(* PLC project benzene-distillation, Generated TextualNotationConverter 1.0 *)
(* stored: creationDateTime 2025-07-30T12:00:00, modificationDateTime 2025-01-30T12:00:00 *)

FUNCTION_BLOCK ANALOG_IN
  VAR_INPUT
    Name : STRING;
    Description : STRING;
    Raw_Signal : REAL;
    PV_High : REAL;
    PV_Low : REAL;
    Scaling_Slope : REAL;
    Scaling_Offset : REAL;
    Alarm_Enable : BOOL;
  END_VAR
  VAR_OUTPUT
    PV : REAL;
    High_Alarm : BOOL;
    Low_Alarm : BOOL;
    General_Fault : BOOL;
  END_VAR

            
          
END_FUNCTION_BLOCK

FUNCTION_BLOCK DIGITAL_IN
  VAR_INPUT
    Name : STRING;
    Description : STRING;
    DI_Raw : BOOL;
    DebounceTime : STRING;
    EnableAlarm : BOOL;
  END_VAR
  VAR_OUTPUT
    DI_Out : BOOL;
    Fault_State : BOOL;
  END_VAR

            
          
END_FUNCTION_BLOCK

FUNCTION_BLOCK PID_BASIC
  VAR_INPUT
    Name : STRING;
    Description : STRING;
    AUTO : BOOL;
    PV : REAL;
    SP : REAL;
    MV_MIN : REAL;
    MV_MAX : REAL;
    X0 : REAL;
    KP : REAL;
    TR : REAL;
    TD : REAL;
    PV_High : REAL;
    PV_Low : REAL;
    Deviation_Limit : REAL;
    Inhibit : BOOL;
  END_VAR
  VAR_OUTPUT
    PV_High_Alarm : BOOL;
    PV_Low_Alarm : BOOL;
    Deviation_Alarm : BOOL;
    XOUT : REAL;
  END_VAR

            
          
END_FUNCTION_BLOCK

FUNCTION_BLOCK VALVE_ELECTRIC
  VAR_INPUT
    Name : STRING;
    Description : STRING;
    Control_Signal : REAL;
    Manual_Mode : BOOL;
    Manual_Position : REAL;
    Open_Limit : REAL;
    Close_Limit : REAL;
    Timeout : STRING;
    Inhibit : BOOL;
  END_VAR
  VAR_OUTPUT
    Valve_Position : REAL;
    Feedback_Pos : REAL;
    Valve_Moving : BOOL;
    Position_Error : BOOL;
    Alarm : BOOL;
  END_VAR

            
          
END_FUNCTION_BLOCK

FUNCTION_BLOCK VALVE_ON_OFF
  VAR_INPUT
    Name : STRING;
    Description : STRING;
    Open_Cmd : BOOL;
    Close_Cmd : BOOL;
    Timeout : STRING;
    Inhibit : BOOL;
  END_VAR
  VAR_OUTPUT
    FB_Opened : BOOL;
    FB_Closed : BOOL;
    Valve_Open_Out : BOOL;
    Valve_Close_Out : BOOL;
    Alarm_Position_Error : BOOL;
    Alarm_General : BOOL;
  END_VAR

            
          
END_FUNCTION_BLOCK

PROGRAM Section2
  VAR
    TE101_Temperature_PV : REAL;
    LIT101_Level_PV : REAL;
    PIT102_Pressure_PV : REAL;
    TIC104_MV_Percent : REAL;
    PV103_Position_FB : REAL;
  END_VAR
  VAR
    TE-101 : ANALOG_IN;
    LIT-101 : ANALOG_IN;
    PIT-102 : ANALOG_IN;
    TIC-104 : PID_BASIC;
    PV-103 : VALVE_ELECTRIC;
    XV-105 : VALVE_ON_OFF;
    LAH-101 : DIGITAL_IN;
    LAL-101 : DIGITAL_IN;
  END_VAR

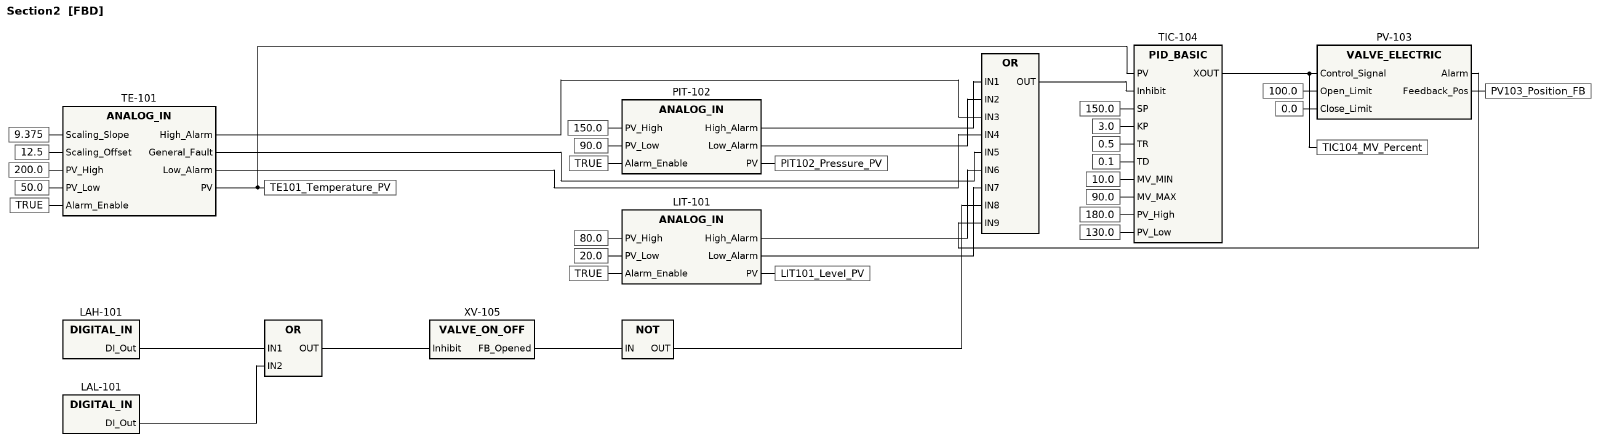
(* FBD diagram, written out as Structured Text *)
LIT-101(PV_High := 80.0, PV_Low := 20.0, Alarm_Enable := TRUE);
LIT101_Level_PV := LIT-101.PV;
PIT-102(PV_High := 150.0, PV_Low := 90.0, Alarm_Enable := TRUE);
PIT102_Pressure_PV := PIT-102.PV;
TE-101(Scaling_Slope := 9.375, Scaling_Offset := 12.5, PV_High := 200.0, PV_Low := 50.0, Alarm_Enable := TRUE);
LAH-101();
LAL-101();
XV-105(Inhibit := LAH-101.DI_Out OR LAL-101.DI_Out);
TIC-104(PV := TE-101.PV, Inhibit := PIT-102.High_Alarm OR PIT-102.Low_Alarm OR TE-101.High_Alarm OR TE-101.Low_Alarm OR TE-101.General_Fault OR LIT-101.High_Alarm OR LIT-101.Low_Alarm OR NOT XV-105.FB_Opened OR PV-103.Alarm, SP := 150.0, KP := 3.0, TR := 0.5, TD := 0.1, MV_MIN := 10.0, MV_MAX := 90.0, PV_High := 180.0, PV_Low := 130.0);
PV-103(Control_Signal := TIC-104.XOUT, Open_Limit := 100.0, Close_Limit := 0.0);
PV103_Position_FB := PV-103.Feedback_Pos;
TE101_Temperature_PV := TE-101.PV;
TIC104_MV_Percent := TIC-104.XOUT;
END_PROGRAM

FUNCTION_BLOCK BOOL_IN
  VAR_INPUT
    Name : STRING;
    Description : STRING;
    Bool_In : BOOL;
    Alarm_OnTrue : BOOL;
    Alarm_OnFalse : BOOL;
    Latch_Enable : BOOL;
    Reset_Latch : BOOL;
  END_VAR
  VAR_OUTPUT
    Bool_Out : BOOL;
    Alarm_Active : BOOL;
    Latched_Status : BOOL;
  END_VAR

            
          
END_FUNCTION_BLOCK

FUNCTION_BLOCK DUTY_STANDBY
  VAR_INPUT
    Name : STRING;
    Description : STRING;
    Enable : BOOL;
    StartRequest : BOOL;
    AlternateEnable : BOOL;
    ForcePumpA : BOOL;
    ForcePumpB : BOOL;
    DutyElapsed : BOOL;
    MinRunElapsed : BOOL;
    SwitchoverDelayElapsed : BOOL;
    StartTimeoutElapsed : BOOL;
    PumpA_RunFB : BOOL;
    PumpB_RunFB : BOOL;
    PumpA_Fault : BOOL;
    PumpB_Fault : BOOL;
    Reset : BOOL;
    Inhibit : BOOL;
  END_VAR
  VAR_OUTPUT
    CmdPumpA : BOOL;
    CmdPumpB : BOOL;
    ActiveIsA : BOOL;
    SwitchedDueToDuty : BOOL;
    SwitchedDueToFailure : BOOL;
    Alarm_FailedStart_A : BOOL;
    Alarm_FailedStart_B : BOOL;
    Alarm_NoAvailablePump : BOOL;
  END_VAR

            
          
END_FUNCTION_BLOCK

FUNCTION_BLOCK MOTOR_2SPD
  VAR_INPUT
    Name : STRING;
    Description : STRING;
    Start_Cmd : BOOL;
    Stop_Cmd : BOOL;
    Speed_High_Cmd : BOOL;
    Speed_Low_Cmd : BOOL;
    Inhibit : BOOL;
  END_VAR
  VAR_OUTPUT
    Motor_Start_Out : BOOL;
    FB_Running : BOOL;
    FB_Trip : BOOL;
    FB_HighSpeed : BOOL;
    FB_LowSpeed : BOOL;
    Alarm_Speed_Error : BOOL;
  END_VAR

            
          
END_FUNCTION_BLOCK

FUNCTION_BLOCK MOTOR_ON_OFF
  VAR_INPUT
    Name : STRING;
    Description : STRING;
    Start_Cmd : BOOL;
    Stop_Cmd : BOOL;
    Start_Delay : STRING;
    MinRunTime : STRING;
    Inhibit : BOOL;
  END_VAR
  VAR_OUTPUT
    Motor_Start_Out : BOOL;
    FB_Running : BOOL;
    FB_Trip : BOOL;
    Alarm_Start_Fail : BOOL;
    Alarm_Stop_Fail : BOOL;
  END_VAR

            
          
END_FUNCTION_BLOCK

FUNCTION_BLOCK MOTOR_VSD
  VAR_INPUT
    Name : STRING;
    Description : STRING;
    Start_Cmd : BOOL;
    Stop_Cmd : BOOL;
    Speed_SP : REAL;
    Accel_Ramp : STRING;
    Decel_Ramp : STRING;
    Inhibit : BOOL;
  END_VAR
  VAR_OUTPUT
    Speed_Out : REAL;
    FB_Running : BOOL;
    FB_Fault : BOOL;
    FB_Ready : BOOL;
    FB_ActualSpeed : REAL;
    Alarm_Speed_Deviation : BOOL;
    Alarm_Comm_Fail : BOOL;
  END_VAR

            
          
END_FUNCTION_BLOCK

FUNCTION_BLOCK RATIO_CONTROL
  VAR_INPUT
    Name : STRING;
    Description : STRING;
    Auto : BOOL;
    PrimaryPV : REAL;
    SecondaryPV : REAL;
    RatioSP : REAL;
    Bias : REAL;
    TrimKp : REAL;
    TrimTi : STRING;
    MV_MIN : REAL;
    MV_MAX : REAL;
    ManOut : REAL;
    Inhibit : BOOL;
  END_VAR
  VAR_OUTPUT
    SlaveSP : REAL;
    ActiveRatio : REAL;
    RatioErr : REAL;
  END_VAR

            
          
END_FUNCTION_BLOCK

FUNCTION_BLOCK SPLIT_RANGE
  VAR_INPUT
    Name : STRING;
    Description : STRING;
    IN : REAL;
    Split_Point : REAL;
    Output1_Start : REAL;
    Output1_End : REAL;
    Output2_Start : REAL;
    Output2_End : REAL;
  END_VAR
  VAR_OUTPUT
    OUT1 : REAL;
    OUT2 : REAL;
  END_VAR

            
          
END_FUNCTION_BLOCK

FUNCTION_BLOCK VOTING_ANALOG
  VAR_INPUT
    Name : STRING;
    Description : STRING;
    Input1 : REAL;
    Input2 : REAL;
    Input3 : REAL;
    Deviation_Limit : REAL;
    Voting_Scheme : STRING;
    EnableAlarm : BOOL;
    Inhibit : BOOL;
  END_VAR
  VAR_OUTPUT
    Voted_Output : REAL;
    Sensor1_Fault : BOOL;
    Sensor2_Fault : BOOL;
    Sensor3_Fault : BOOL;
    Alarm_Voting_Error : BOOL;
    Healthy_Sensors_Count : INT;
  END_VAR

            
          
END_FUNCTION_BLOCK

PROGRAM Section3
  VAR
    Reboiler_Temperature_PV_TI106 : REAL;
    Steam_Flow_PV_FIT101 : REAL;
    Column_Pressure_PV_PT101 : REAL;
    FIC104_MV_SteamValveCmd : REAL;
    LIC002_LowLevel_Trip : BOOL;
  END_VAR
  VAR
    TI-106 : ANALOG_IN;
    FIT-101 : ANALOG_IN;
    PT-101 : ANALOG_IN;
    FIC-104 : PID_BASIC;
    TCV-106 : VALVE_ELECTRIC;
    LIC-002 : BOOL_IN;
    TAH-106 : BOOL_IN;
    TAL-106 : BOOL_IN;
    FAH-104 : BOOL_IN;
  END_VAR
  VAR  (* added by the conversion: wires and edge detectors of the diagram *)
    _OR38_OUT : BOOL;
  END_VAR

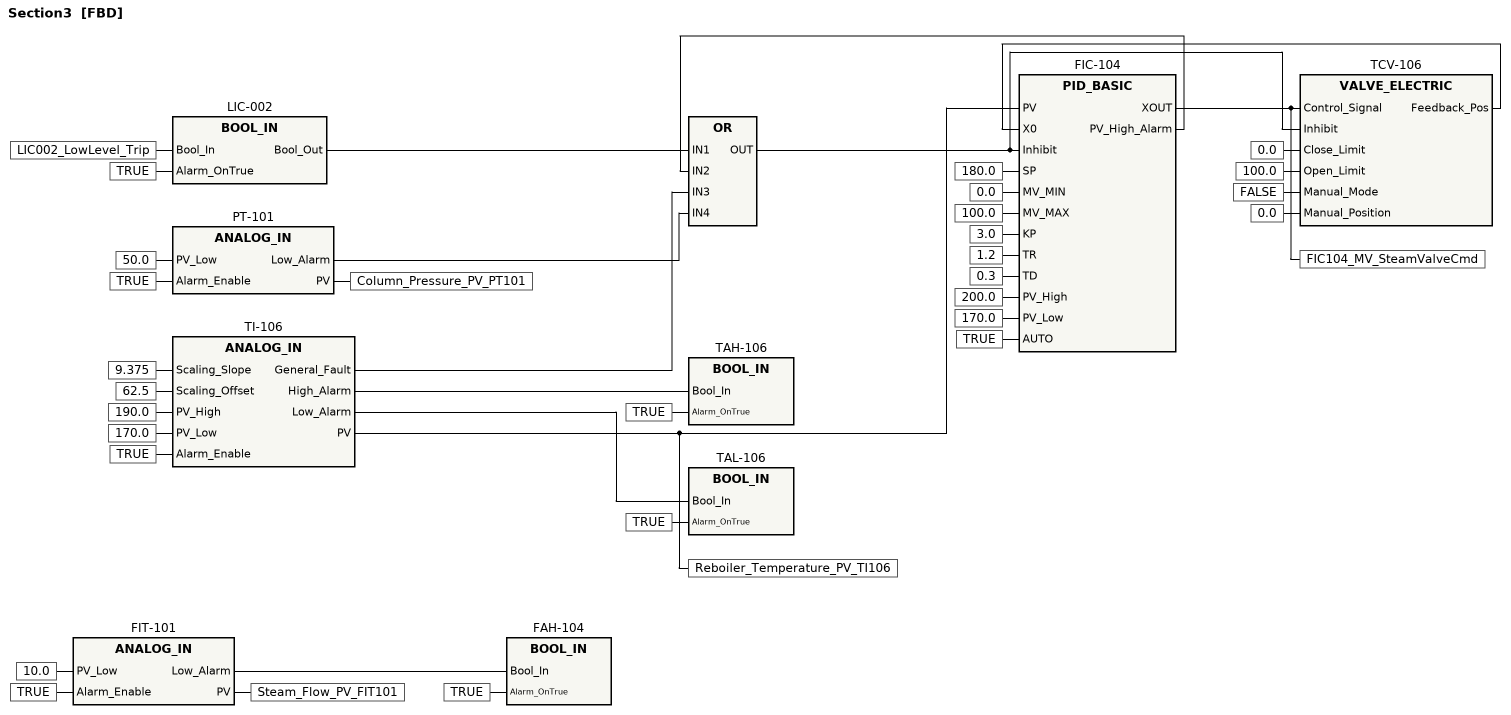
(* FBD diagram, written out as Structured Text *)
PT-101(PV_Low := 50.0, Alarm_Enable := TRUE);
Column_Pressure_PV_PT101 := PT-101.PV;
TI-106(Scaling_Slope := 9.375, Scaling_Offset := 62.5, PV_High := 190.0, PV_Low := 170.0, Alarm_Enable := TRUE);
LIC-002(Bool_In := LIC002_LowLevel_Trip, Alarm_OnTrue := TRUE);
_OR38_OUT := LIC-002.Bool_Out OR FIC-104.PV_High_Alarm OR TI-106.General_Fault OR PT-101.Low_Alarm;
TCV-106(Control_Signal := FIC-104.XOUT, Inhibit := _OR38_OUT, Close_Limit := 0.0, Open_Limit := 100.0, Manual_Mode := FALSE, Manual_Position := 0.0);
FIC-104(PV := TI-106.PV, X0 := TCV-106.Feedback_Pos, Inhibit := _OR38_OUT, SP := 180.0, MV_MIN := 0.0, MV_MAX := 100.0, KP := 3.0, TR := 1.2, TD := 0.3, PV_High := 200.0, PV_Low := 170.0, AUTO := TRUE);
FIC104_MV_SteamValveCmd := FIC-104.XOUT;
Reboiler_Temperature_PV_TI106 := TI-106.PV;
FIT-101(PV_Low := 10.0, Alarm_Enable := TRUE);
Steam_Flow_PV_FIT101 := FIT-101.PV;
TAH-106(Bool_In := TI-106.High_Alarm, Alarm_OnTrue := TRUE);
TAL-106(Bool_In := TI-106.Low_Alarm, Alarm_OnTrue := TRUE);
FAH-104(Bool_In := FIT-101.Low_Alarm, Alarm_OnTrue := TRUE);
END_PROGRAM

PROGRAM Section4
  VAR
    LT_105_Level_PV : REAL;
    FT_107_Flow_PV : REAL;
    PT_104_Pressure_PV : REAL;
    LIC_104_RSP_to_FIC_107_GPM : REAL;
    FIC_107_Control_Signal_to_LV_107 : REAL;
    XV103_NotOpen : BOOL;
    Cascade_Inhibit : BOOL;
    Permissive_OK : BOOL;
  END_VAR
  VAR
    LT-105 : ANALOG_IN;
    FT-107 : ANALOG_IN;
    PT-104 : ANALOG_IN;
    LIC-104 : PID_BASIC;
    FIC-107 : PID_BASIC;
    PIC-104 : PID_BASIC;
    LV-107 : VALVE_ELECTRIC;
    XV-103 : VALVE_ON_OFF;
  END_VAR
  VAR  (* added by the conversion: wires and edge detectors of the diagram *)
    _NOT80_OUT : BOOL;
    _OR79_OUT : BOOL;
    _MULT83_OUT : REAL;
  END_VAR

(* FBD diagram, written out as Structured Text *)
XV-103();
_NOT80_OUT := NOT XV-103.FB_Opened;
LT-105(PV_High := 90.0, PV_Low := 10.0, Alarm_Enable := TRUE);
PT-104(PV_High := 30.0, PV_Low := 15.0, Alarm_Enable := TRUE);
FT-107(PV_High := 50.0, PV_Low := 0.0, Alarm_Enable := TRUE);
LIC-104(PV := LT-105.PV, Inhibit := _OR79_OUT, AUTO := TON(NOT _OR79_OUT, T#30s), SP := 65.0, KP := 1.5, TR := 2.5, TD := 0.0, MV_MIN := 0.0, MV_MAX := 100.0, X0 := 40.0, PV_High := 90.0, PV_Low := 10.0);
_MULT83_OUT := MULT(LIC-104.XOUT, 0.5);
FIC-107(SP := _MULT83_OUT, PV := FT-107.PV, Inhibit := _OR79_OUT, AUTO := NOT _OR79_OUT, KP := 4.0, TR := 0.5, TD := 0.0, MV_MIN := 0.0, MV_MAX := 100.0, PV_High := 50.0, PV_Low := 0.0);
LV-107(Control_Signal := FIC-107.XOUT, Inhibit := PT-104.High_Alarm, Manual_Mode := PT-104.High_Alarm, Open_Limit := 100.0, Close_Limit := 0.0, Manual_Position := 0.0);
_OR79_OUT := _NOT80_OUT OR LT-105.Low_Alarm OR PT-104.Low_Alarm OR PT-104.High_Alarm OR FT-107.General_Fault OR LV-107.Alarm;
Cascade_Inhibit := _OR79_OUT;
FIC_107_Control_Signal_to_LV_107 := FIC-107.XOUT;
FT_107_Flow_PV := FT-107.PV;
LIC_104_RSP_to_FIC_107_GPM := _MULT83_OUT;
LT_105_Level_PV := LT-105.PV;
PT_104_Pressure_PV := PT-104.PV;
Permissive_OK := NOT _OR79_OUT;
XV103_NotOpen := _NOT80_OUT;
PIC-104(PV := PT-104.PV);
END_PROGRAM

PROGRAM Section5
  VAR
    FI102_FlowRate : REAL;
    PI102_Pressure : REAL;
    LCV102_PositionCmd : REAL;
    XV102A_OpenCmd : BOOL;
    XV102A_CloseCmd : BOOL;
    XV102B_OpenCmd : BOOL;
    XV102B_CloseCmd : BOOL;
    XV102A_OpenFB : BOOL;
    XV102B_OpenFB : BOOL;
    P102A_MotorStart_Out : BOOL;
    P102B_MotorStart_Out : BOOL;
    LIC102_LevelPermissive_OK : BOOL;
    LIC102_LevelPermissiveIn : BOOL;
  END_VAR
  VAR
    FI-102 : ANALOG_IN;
    PI-102 : ANALOG_IN;
    LCV-102 : VALVE_ELECTRIC;
    XV-102A : VALVE_ON_OFF;
    XV-102B : VALVE_ON_OFF;
    P-102A_MotorFault : DIGITAL_IN;
    P-102B_MotorFault : DIGITAL_IN;
    LIC-102_LevelPermissive : BOOL_IN;
    P-102A : MOTOR_ON_OFF;
    P-102B : MOTOR_ON_OFF;
    P-102_DutyStandby : DUTY_STANDBY;
    LowPressure10s_TON : TON;
    SwitchoverDelay5s_TON : TON;
    MinRun30m_TON : TON;
    SuctionBypass10s_TON : TON;
  END_VAR
  VAR  (* added by the conversion: wires and edge detectors of the diagram *)
    _OR133_OUT : BOOL;
    _OR134_OUT : BOOL;
    _AND154_OUT : BOOL;
  END_VAR

(* FBD diagram, written out as Structured Text *)
FI-102(PV_High := 700.0, PV_Low := 500.0, Alarm_Enable := TRUE);
FI102_FlowRate := FI-102.PV;
P-102A_MotorFault();
PI-102(PV_Low := 25.0, Alarm_Enable := TRUE);
LowPressure10s_TON(IN := PI-102.Low_Alarm, PT := T#10s);
_OR133_OUT := P-102A_MotorFault.DI_Out OR P-102_DutyStandby.ActiveIsA AND LowPressure10s_TON.Q;
P-102B_MotorFault();
_OR134_OUT := P-102B_MotorFault.DI_Out OR NOT P-102_DutyStandby.ActiveIsA AND LowPressure10s_TON.Q;
SwitchoverDelay5s_TON(IN := _OR133_OUT OR _OR134_OUT, PT := T#5s);
XV-102A();
SuctionBypass10s_TON(IN := P-102_DutyStandby.SwitchedDueToFailure, PT := T#10s);
_AND154_OUT := NOT (PI-102.PV > 15.0) AND NOT SuctionBypass10s_TON.Q;
LIC-102_LevelPermissive(Bool_In := LIC102_LevelPermissiveIn, Alarm_OnFalse := TRUE);
P-102A(Start_Cmd := P-102_DutyStandby.CmdPumpA OR FI-102.High_Alarm, Inhibit := NOT XV-102A.FB_Opened OR XV-102A.Alarm_Position_Error OR XV-102A.Alarm_General OR _AND154_OUT OR P-102A_MotorFault.DI_Out OR LIC-102_LevelPermissive.Alarm_Active, MinRunTime := T#30m);
XV-102B();
P-102B(Start_Cmd := P-102_DutyStandby.CmdPumpB OR FI-102.High_Alarm, Inhibit := NOT XV-102B.FB_Opened OR XV-102B.Alarm_Position_Error OR XV-102B.Alarm_General OR _AND154_OUT OR P-102B_MotorFault.DI_Out OR LIC-102_LevelPermissive.Alarm_Active, MinRunTime := T#30m);
MinRun30m_TON(IN := P-102A.FB_Running OR P-102B.FB_Running, PT := T#30m);
P-102_DutyStandby(SwitchoverDelayElapsed := SwitchoverDelay5s_TON.Q, PumpA_RunFB := P-102A.FB_Running, PumpB_RunFB := P-102B.FB_Running, PumpA_Fault := _OR133_OUT, PumpB_Fault := _OR134_OUT, MinRunElapsed := MinRun30m_TON.Q, Enable := TRUE, StartRequest := TRUE, AlternateEnable := FALSE);
LCV-102(Inhibit := P-102_DutyStandby.Alarm_NoAvailablePump);
LCV102_PositionCmd := LCV-102.Valve_Position;
LIC102_LevelPermissive_OK := LIC-102_LevelPermissive.Bool_Out;
P102A_MotorStart_Out := P-102A.Motor_Start_Out;
P102B_MotorStart_Out := P-102B.Motor_Start_Out;
PI102_Pressure := PI-102.PV;
XV102A_CloseCmd := XV-102A.Valve_Close_Out;
XV102A_OpenCmd := XV-102A.Valve_Open_Out;
XV102A_OpenFB := XV-102A.FB_Opened;
XV102B_CloseCmd := XV-102B.Valve_Close_Out;
XV102B_OpenCmd := XV-102B.Valve_Open_Out;
XV102B_OpenFB := XV-102B.FB_Opened;
END_PROGRAM

PROGRAM Section6
  VAR
    FT105_FeedFlowRate : REAL;
    FT106_BottomsFlowRate : REAL;
    FT106_SP_From_IIC104 : REAL;
    LIC002_LevelPV : REAL;
  END_VAR
  VAR
    FT-105 : ANALOG_IN;
    FT-106 : ANALOG_IN;
    FV-101 : VALVE_ELECTRIC;
    IIC-104 : RATIO_CONTROL;
    FIC-106 : PID_BASIC;
    LIC-002 : PID_BASIC;
    LIC-002-LOW_LEVEL_ILK : BOOL_IN;
    FEED_PUMP_RUN : DIGITAL_IN;
    BOTTOMS_PUMP_RUN : DIGITAL_IN;
  END_VAR
  VAR  (* added by the conversion: wires and edge detectors of the diagram *)
    _GT199_OUT : BOOL;
    _OR202_OUT : BOOL;
  END_VAR

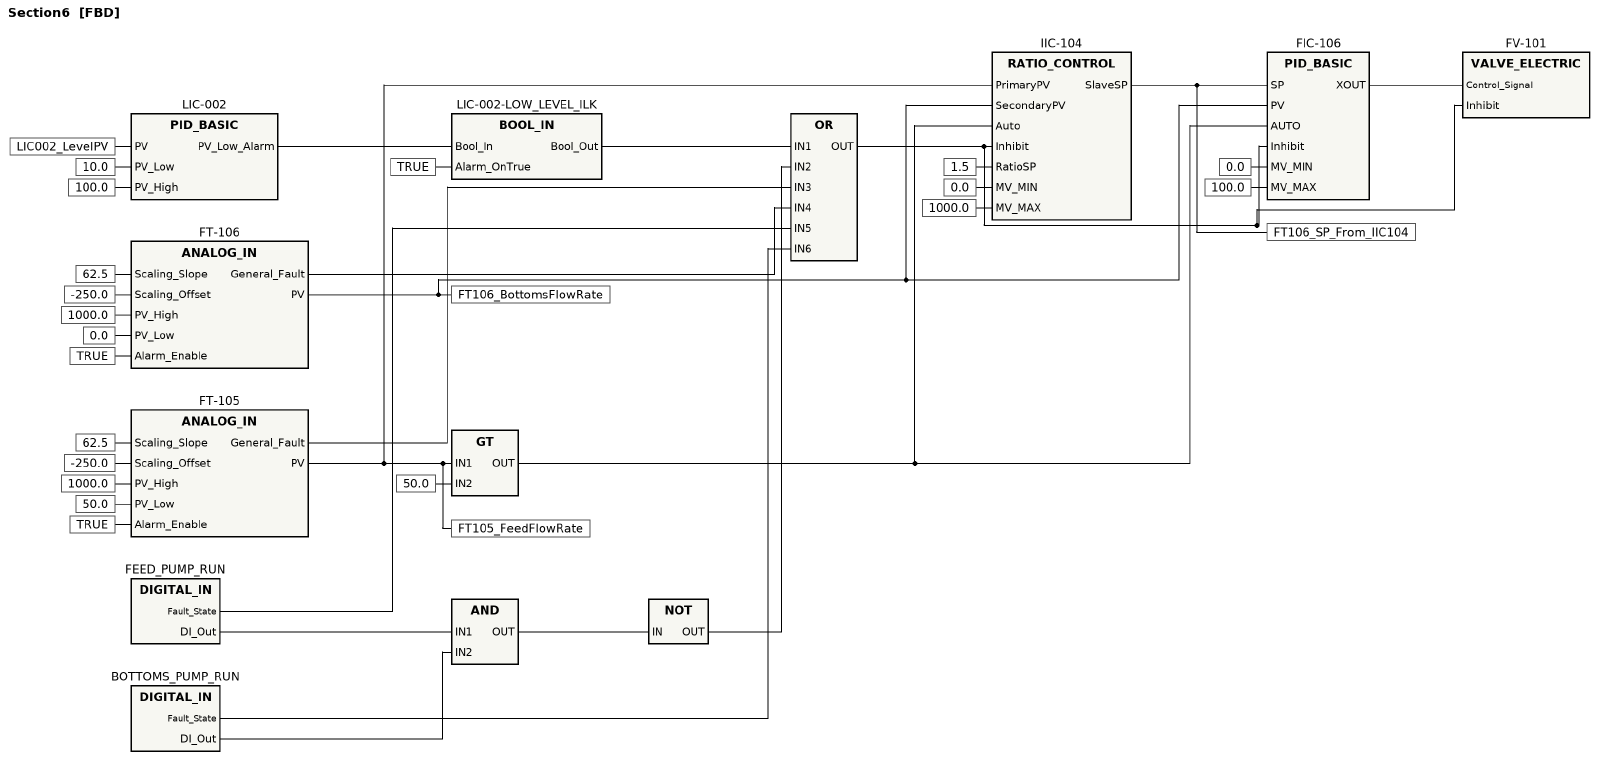
(* FBD diagram, written out as Structured Text *)
FT-105(Scaling_Slope := 62.5, Scaling_Offset := -250.0, PV_High := 1000.0, PV_Low := 50.0, Alarm_Enable := TRUE);
FT105_FeedFlowRate := FT-105.PV;
FT-106(Scaling_Slope := 62.5, Scaling_Offset := -250.0, PV_High := 1000.0, PV_Low := 0.0, Alarm_Enable := TRUE);
FT106_BottomsFlowRate := FT-106.PV;
_GT199_OUT := FT-105.PV > 50.0;
LIC-002(PV := LIC002_LevelPV, PV_Low := 10.0, PV_High := 100.0);
LIC-002-LOW_LEVEL_ILK(Bool_In := LIC-002.PV_Low_Alarm, Alarm_OnTrue := TRUE);
FEED_PUMP_RUN();
BOTTOMS_PUMP_RUN();
_OR202_OUT := LIC-002-LOW_LEVEL_ILK.Bool_Out OR NOT (FEED_PUMP_RUN.DI_Out AND BOTTOMS_PUMP_RUN.DI_Out) OR FT-105.General_Fault OR FT-106.General_Fault OR FEED_PUMP_RUN.Fault_State OR BOTTOMS_PUMP_RUN.Fault_State;
IIC-104(PrimaryPV := FT-105.PV, SecondaryPV := FT-106.PV, Auto := _GT199_OUT, Inhibit := _OR202_OUT, RatioSP := 1.5, MV_MIN := 0.0, MV_MAX := 1000.0);
FT106_SP_From_IIC104 := IIC-104.SlaveSP;
FIC-106(SP := IIC-104.SlaveSP, PV := FT-106.PV, AUTO := _GT199_OUT, Inhibit := _OR202_OUT, MV_MIN := 0.0, MV_MAX := 100.0);
FV-101(Control_Signal := FIC-106.XOUT, Inhibit := _OR202_OUT);
END_PROGRAM

CONFIGURATION Config0
  RESOURCE Res0 ON PLC
    TASK task0(INTERVAL := T#20ms, PRIORITY := 0);
    PROGRAM instance0 WITH task0 : Section2;
    PROGRAM instance_1 WITH task0 : Section3;
    PROGRAM instance_2 WITH task0 : Section4;
    PROGRAM instance_3 WITH task0 : Section5;
    PROGRAM instance_4 WITH task0 : Section6;
  END_RESOURCE
END_CONFIGURATION
